// TwinCAT 3 PLC project PLC_Projects
// ProgramVersion: 3.1.4024.0
// libraries:
//   Tc2_MC2, * (Beckhoff Automation GmbH)
//   Tc2_MC2_XFC, * (Beckhoff Automation GmbH)
//   Tc2_Standard, * (Beckhoff Automation GmbH)
//   Tc2_System, * (Beckhoff Automation GmbH)
//   Tc3_Module, * (Beckhoff Automation GmbH)
// project tree:
//   / PlcTask.TcTTO
//   POUs/ MAIN.TcPOU
// real-time tasks:
//   TASK PlcTask: cycle T#500us, priority 20, ADS port 350
// motion (NC):
//   TASK NC-Task 1 SAF: cycle T#500us, priority 4, ADS port 501
//   TASK NC-Task 1 SVB: cycle T#1ms, priority 8, ADS port 511
//   AXIS EncodeAxis (id 1)
//     General: UnitFlags=#x00000004
//     OtherSettings: AllowMotionCmdToSlave=true
//     encoder EncType=4
//       EncPara: ScaleFactorNumerator=1, ModuloFactor=100, MaxCount=#xffffffff
//         Inc: RefSoftSyncMask=#x0000ffff
//     drive DrvType=5
//       Analog: TorqueSetpointScale=10, ScaleFactorActTorque=0.1
//       TimeComp: TaskDelayCycles=1
//     controller CtrType=1
//       CtrPara: PriorControlFactor=1
//         Observer: BandWidth=20
//   AXIS SimulationAxis (id 2)
//     General: UnitName=Degree, UnitFlags=#x00000004
//     Dynamic: Acceleration=14535, Deceleration=14535, Jerk=43605
//     Velo: RefSearch=96.9, RefSync=96.9, SlowManual=484.5, FastManual=2907, Fast=9690, Maximum=9690
//     OtherSettings: AllowMotionCmdToSlave=true
//     encoder EncType=1
//       EncPara: ScaleFactorNumerator=360, ScaleFactorDenominator=1048576
//     drive DrvType=5
//       Analog: VeloReferenz=10659, TorqueSetpointScale=10, ScaleFactorActTorque=0.1
//       TimeComp: TaskDelayCycles=1
//     controller CtrType=1
//       CtrPara: PriorControlFactor=1
//         PosDiffControl: Enable=false
//         Observer: BandWidth=20
// I/O:
//   DEVICE Device 4 (EtherCAT), AmsNetId 5.131.180.184.5.1
//     Term 2 (EK1100) [EK1100 EtherCAT Coupler (2A E-Bus)]
//       Term 3 (EL5101) [EL5101 1Ch. Inc. Encoder 5V]
//       Term 4 (EL2252) [EL2252 2Ch. Dig. Output 24V, 0.5A, DC Time Stamp]
//       Term 5 (EL1252) [EL1252 2Ch. Fast Dig. Input 24V, 1µs, DC Latch]
//       Term 5 (EL9011) [EL9011 End Terminal]
// variable links:
//   NC-Task 1 SAF/Axes/EncodeAxis <-> Device 4 (EtherCAT)/Term 2 (EK1100)/Term 3 (EL5101)
//     Enc/Inputs/In/nDataIn1 <-> ENC Status/Counter value
//     Enc/Inputs/In/nDataIn2 <-> ENC Status/Latch value
//     Enc/Inputs/In/nState1 @bit 4 <-> ENC Status/Status/Counter overflow
//     Enc/Inputs/In/nState1 @bit 3 <-> ENC Status/Status/Counter underflow
//     Enc/Inputs/In/nState1 @bit 7 <-> ENC Status/Status/Extrapolation stall
//     Enc/Inputs/In/nState1 <-> ENC Status/Status/Latch C valid
//     Enc/Inputs/In/nState1 @bit 1 <-> ENC Status/Status/Latch extern valid
//     Enc/Inputs/In/nState1 @bit 6 <-> ENC Status/Status/Open circuit
//     Enc/Inputs/In/nState1 @bit 2 <-> ENC Status/Status/Set counter done
//     Enc/Inputs/In/nState1 @bit 5 <-> ENC Status/Status/Status of input status
//     Enc/Inputs/In/nState2 @bit 4 <-> ENC Status/Status/Status of extern latch
//     Enc/Inputs/In/nState2 <-> ENC Status/Status/Status of input A
//     Enc/Inputs/In/nState2 @bit 1 <-> ENC Status/Status/Status of input B
//     Enc/Inputs/In/nState2 @bit 2 <-> ENC Status/Status/Status of input C
//     Enc/Inputs/In/nState2 @bit 3 <-> ENC Status/Status/Status of input gate
//     Enc/Inputs/In/nState2 @bit 5 <-> ENC Status/Status/Sync error
//     Enc/Inputs/In/nState2 @bit 6 <-> ENC Status/Status/TxPDO State
//     Enc/Inputs/In/nState2 @bit 7 <-> ENC Status/Status/TxPDO Toggle
//     Enc/Inputs/In/nState4 @bit 1 <-> WcState/InputToggle
//     Enc/Inputs/In/nState4 <-> WcState/WcState
//     Enc/Outputs/Out/nCtrl1 <-> ENC Control/Control/Enable latch C
//     Enc/Outputs/Out/nCtrl1 @bit 3 <-> ENC Control/Control/Enable latch extern on negative edge
//     Enc/Outputs/Out/nCtrl1 @bit 1 <-> ENC Control/Control/Enable latch extern on positive edge
//     Enc/Outputs/Out/nCtrl1 @bit 2 <-> ENC Control/Control/Set counter
//     Enc/Outputs/Out/nDataOut1 <-> ENC Control/Set counter value
//   PLC_Projects/PLC_Projects Instance <-> Device 4 (EtherCAT)/Term 2 (EK1100)/Term 4 (EL2252)
//     PlcTask Outputs/MAIN.EL2252.Activate <-> DC Sync Activate/Activate
//     PlcTask Outputs/MAIN.EL2252.Output1 <-> Channel 1/Output
//     PlcTask Outputs/MAIN.EL2252.Output2 <-> Channel 2/Output
//     PlcTask Outputs/MAIN.EL2252.StartTime <-> DC Sync Start/StartTime
//     PlcTask Outputs/MAIN.EL2252.TriState1 <-> Channel 1/TriState
//     PlcTask Outputs/MAIN.EL2252.TriState2 <-> Channel 2/TriState
//   PLC_Projects/PLC_Projects Instance <-> Device 4 (EtherCAT)/Term 2 (EK1100)/Term 5 (EL1252)
//     PlcTask Inputs/MAIN.input1 <-> Channel 1/Input
//     PlcTask Inputs/MAIN.input2 <-> Channel 2/Input
//   PLC_Projects/PLC_Projects Instance <-> NC-Task 1 SAF/Axes/EncodeAxis
//     PlcTask Inputs/MAIN.stEncodeAxisReference.NcToPlc <-> Outputs/ToPlc
//     PlcTask Outputs/MAIN.stEncodeAxisReference.PlcToNc <-> Inputs/FromPlc
//   PLC_Projects/PLC_Projects Instance <-> NC-Task 1 SAF/Axes/SimulationAxis
//     PlcTask Inputs/MAIN.stSimAxisReference.NcToPlc <-> Outputs/ToPlc
//     PlcTask Outputs/MAIN.stSimAxisReference.PlcToNc <-> Inputs/FromPlc

CONFIGURATION PLC_Projects
    RESOURCE PLC ON TwinCAT3
        TASK PlcTask(INTERVAL := T#500us, PRIORITY := 20);
        PROGRAM MAIN WITH PlcTask : MAIN;
    END_RESOURCE
END_CONFIGURATION

// ---- POUs/MAIN.TcPOU
PROGRAM MAIN
VAR
   
    useSimulationAxis: BOOL; //Switch Axis
    bSetEncoderPos: BOOL; //Set Encode Pos to Zero
    bEnableCamOutput: BOOL := TRUE; //Start XFC Output Cam
    
    stEncodeAxisReference : AXIS_REF;
	encoderPosition: LREAL;
    fbSetEncoderPosition : MC_SetPosition;
	encodeSetPos: LREAL;
	fbDigitalCam: MC_DigitalCamSwitch;
    stCamSwitchOptions : ST_CamSwitchOptions;
    CamSwitchData : ARRAY[0..2] OF MC_CamSwitch;
    CamSwitchRef   : CAMSWITCH_REF;
    EL2252_Out1_Ref : OUTPUT_REF;
    EL2252_Out2_Ref : OUTPUT_REF;
    TrackOptions : TRACK_REF;
	fbEL2252: XFC_EL2252_V2;
    EL2252_Channel1_TrackOptions    : TRACK_REF;
    EL2252_Channel2_TrackOptions    : TRACK_REF;
    EL2252        : EL2252_IoInterface;
    stSimAxisReference : AXIS_REF;
    input1 AT %I* : BOOL;
    input2 AT %I* : BOOL;
	fbTest: MC_Power;
    stAxisReference : AXIS_REF;

END_VAR

(* ----------------- Encoder---------------------------------------------------- *)

(* Steps 
1.Set Axis as Simulation Axis
2.In Endcoder -> Go to NC-EncodeTab -> Link you Encode as per the type
3.Then Set Num & Den Factor according
    Encode 1 Pulse = 1 MM then keep Num = 1 & Den = 1 
*)

//Encoder Position
encoderPosition := stEncodeAxisReference.NcToPlc.ModuloActPos;

//Set Encoder Position
fbSetEncoderPosition(
	Axis:=stEncodeAxisReference, 
	Execute:=bSetEncoderPos, 
	Position:=encodeSetPos, 
	Mode:= , 
	Options:= , 
	Done=> , 
	Busy=> , 
	Error=> , 
	ErrorID=> );
bSetEncoderPos := FALSE;

(*-------------------------------------------------------------------------------*)

(* ----------------- Simulation Axis Enable ------------------------------------ *)

fbTest(
	Axis:=stSimAxisReference, 
	Enable:=1, 
	Enable_Positive:=1, 
	Enable_Negative:=1, 
	Override:=100, 
	BufferMode:= , 
	Options:= , 
	Status=> , 
	Busy=> , 
	Active=> , 
	Error=> , 
	ErrorID=> );
  
(*-------------------------------------------------------------------------------*)


(* ----------------- Simulation Axis Enable ------------------------------------ *)
IF useSimulationAxis THEN
    stAxisReference := stSimAxisReference;
ELSE
    stAxisReference := stEncodeAxisReference;
END_IF

(*-------------------------------------------------------------------------------*)
    
(* ----------------- Output Switching ------------------------------------------ *)

//Cam Options
stCamSwitchOptions.EncoderIndex := 0;
stCamSwitchOptions.UseAcceleration := 0;

//Cam Swith Data 1 
CamSwitchData[0].AxisDirection := E_CamSwitchDirection.CAMSWITCHDIRECTION_POSITIVE;
CamSwitchData[0].CamSwitchMode := E_CamSwitchMode.CAMSWITCHMODE_POSITION;
IF useSimulationAxis THEN
    CamSwitchData[0].FirstOnPosition := 60.0;
    CamSwitchData[0].LastOnPosition := 65.0;
ELSE
    CamSwitchData[0].FirstOnPosition := 20.0;
    CamSwitchData[0].LastOnPosition := 25.0;
END_IF
//CamSwitchData[0].Duration := ;

//Cam Swith Data 2 
CamSwitchData[1].AxisDirection := E_CamSwitchDirection.CAMSWITCHDIRECTION_POSITIVE;
CamSwitchData[1].CamSwitchMode := E_CamSwitchMode.CAMSWITCHMODE_POSITION;
IF useSimulationAxis THEN
    CamSwitchData[1].FirstOnPosition := 150.0;
    CamSwitchData[1].LastOnPosition := 160.0;
ELSE
    CamSwitchData[1].FirstOnPosition := 50.0;
    CamSwitchData[1].LastOnPosition := 55.0;
END_IF
//CamSwitchData[0].Duration := ;

//Cam Swith Data 3 
CamSwitchData[2].AxisDirection := E_CamSwitchDirection.CAMSWITCHDIRECTION_POSITIVE;
CamSwitchData[2].CamSwitchMode := E_CamSwitchMode.CAMSWITCHMODE_POSITION;
IF useSimulationAxis THEN
    CamSwitchData[2].FirstOnPosition := 300.0;
    CamSwitchData[2].LastOnPosition := 310.0;
ELSE
    CamSwitchData[2].FirstOnPosition := 80.0;
    CamSwitchData[2].LastOnPosition := 85.0;
END_IF
//CamSwitchData[0].Duration := ;

//Track Options
TrackOptions.ModuloPositions := TRUE;

IF useSimulationAxis THEN
    TrackOptions.ModuloFactor := 360;
ELSE
     TrackOptions.ModuloFactor := 100; 
END_IF

//Cam Switch Reference
CamSwitchRef.NumberOfSwitches := 3;
CamSwitchRef.pSwitches        := ADR(CamSwitchData);
CamSwitchRef.SizeOfSwitches   := SIZEOF(CamSwitchData);

//Digital Cam
fbDigitalCam(
	Axis:=stAxisReference,  
	Switches:=CamSwitchRef, 
	Output:=EL2252_Out1_Ref, 
	TrackOptions:=TrackOptions, 
	Enable:=bEnableCamOutput, 
	Options:= , 
	InOperation=> , 
	Busy=> , 
	Error=> , 
	ErrorID=> );

//EL2252 Output 
fbEL2252(
	ForceWhenLate:=0, 
	Error=> , 
	ErrorID=> , 
	ErrorOutputMissed=> , 
	PrecisionReduced=> , 
	Output1:=EL2252_Out1_Ref, 
	Output2:=EL2252_Out2_Ref, 
	TrackOptions1:=TrackOptions, 
	TrackOptions2:=EL2252_Channel2_TrackOptions, 
	EL2252:=EL2252);

(*-------------------------------------------------------------------------------*)

END_PROGRAM
